# EPICS substitutions: iocBoot/ioczzz/pseudoMotor.substitutions
# Pseudo-motors
# Note: This databases will be in the next release of motor, not in zzzApp

# This is a simple example using the sumDiff2D database.  This takes 2 real motors and makes 2 soft motors,
# SUM which moves both motors together, and DIFF which moves them in opposite directions.
# It can be used for slits, for K/B mirror benders, etc.

file "$(MOTOR)/motorApp/Db/pseudoMotor.db"
{
pattern
{P,       M,           DINP,                        OUT,                     RDBL,                          STOO,     DESC, EGU, DIR, VELO, VBAS, ACCL, BDST, BVEL,                    BACC, MRES,   RRES, PREC,  DHLM, DLLM}
{zzz:,  pm1, "zzz:KBV:Done NPP NMS", "zzz:pm1DVAL.VAL PP MS", "zzz:KBV:Readback.G NPP NMS", "zzz:KBV:Stop PP MS",    "Vert. curvature",          mm,  Pos,   1,    .1,   .1,    0,    1,   .1, .1,     1.0,  3,    10000, -10000}
{zzz:,  pm2, "zzz:KBV:Done NPP NMS", "zzz:pm2DVAL.VAL PP MS", "zzz:KBV:Readback.H NPP NMS", "zzz:KBV:Stop PP MS",    "Vert. Ellipticity",        mm,  Pos,   1,    .1,   .1,    0,    1,   .1, .1,     1.0,  3,    10000, -10000}
{zzz:,  pm3, "zzz:KBH:Done NPP NMS", "zzz:pm3DVAL.VAL PP MS", "zzz:KBH:Readback.G NPP NMS", "zzz:KBH:Stop PP MS",    "Hor. curvature",          mm,  Pos,   1,    .1,   .1,    0,    1,   .1, .1,     1.0,  3,    10000, -10000}
{zzz:,  pm4, "zzz:KBH:Done NPP NMS", "zzz:pm4DVAL.VAL PP MS", "zzz:KBH:Readback.H NPP NMS", "zzz:KBH:Stop PP MS",    "Hor. ellipticity",        mm,  Pos,   1,    .1,   .1,    0,    1,   .1, .1,     1.0,  3,    10000, -10000}
}

file "$(MOTOR)/motorApp/Db/sumDiff2D.db"
{
pattern
{P,      T,   SUM, DIFF,     M1DRV,    M1RBV,   M2DRV,   M2RBV,   M1STOP,   M1DONE,   M2STOP,   M2DONE,  PREC}
{zzz:, KBV:,  pm1,  pm2,    m1.VAL,   m1.RBV,  m2.VAL,  m2.RBV,  m1.STOP,  m1.DMOV,  m2.STOP,  m2.DMOV,    1}
{zzz:, KBH:,  pm3,  pm4,    m3.VAL,   m3.RBV,  m4.VAL,  m4.RBV,  m3.STOP,  m3.DMOV,  m4.STOP,  m4.DMOV,    1}
}
